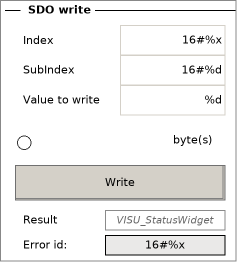
VISUALIZATION VISU_FaulhaberDrive_SDOWrite  // 237x262
VAR_IN_OUT
	drive : FaulhaberDrive;
    widget : FaulhaberDriveWidget;
END_VAR
    Textfield (120,85 105x30), "%d", text variable: drive.processes.write.set.value4Bytes, invisible if: widget.writeNoOfBytes <> 4, input disabled if: drive.processes.write.statuses.enabledStatus.disabled
        OnMouseClick: write the text variable via VisuDialogs.Numpad
    Textfield (120,85 105x30), "%d", text variable: drive.processes.write.set.value2Bytes, invisible if: widget.writeNoOfBytes <> 2, input disabled if: drive.processes.write.statuses.enabledStatus.disabled
        OnMouseClick: write the text variable via VisuDialogs.Numpad
    Textfield (120,85 105x30), "%d", text variable: drive.processes.write.set.value1Byte, invisible if: widget.writeNoOfBytes <> 1, input disabled if: drive.processes.write.statuses.enabledStatus.disabled
        OnMouseClick: write the text variable via Default
    Label (20,26 100x29), "Index"
    Button (15,165 210x35), "Write", input disabled if: drive.processes.write.statuses.enabledStatus.disabled
        OnMouseClick: execute { drive.processes.write.set.noOfBytes := widget.writeNoOfBytes; drive.processes.write.do_request := TRUE; }
    Textfield (120,55 105x30), "16#%d", text variable: drive.processes.write.set.subindex, input disabled if: drive.processes.write.statuses.enabledStatus.disabled
        OnMouseClick: write the text variable via Default
    Label (20,55 95x30), "SubIndex"
    Line (5,10) (20,10)
    Label (25,0 150x20), "SDO write"
    Line (95,10) (235,10)
    Textfield (120,25 105x30), "16#%x", text variable: drive.processes.write.set.index, input disabled if: drive.processes.write.statuses.enabledStatus.disabled
        OnMouseClick: write the text variable via Default
    Frame (105,210 120x20)
        shows VISU_StatusWidget(widget := widget.sdoWriteStatus)
    RadioButton (15,125 155x35), variable: widget.writeNoOfBytesRadioButtonItem, input disabled if: drive.processes.write.statuses.enabledStatus.disabled
        Areas[0]: Text=1
        Areas[1]: Text=2
        Areas[2]: Text=4
    Label (170,125 55x30), "byte(s)"
    Label (20,205 80x30), "Result"
    Rectangle (105,235 120x20), "16#%x", text variable: drive.processes.write.errorId
    Label (20,230 80x30), "Error id:"
    Label (20,85 100x30), "Value to write"
END_VISUALIZATION

(* stored: Version 1.1.0.1, ProductVersion 3.1.4019.2
   Visu VISU_FaulhaberDrive_SDOWrite: Id {5ba5cd2c-a076-4ce2-8d2c-343128275525} *)
